{attribute 'linkalways'} 
{attribute 'no_explicit_call' := 'This FB is a CLASS and must be accessed using methods or properties'}
{attribute 'enable_dynamic_creation'}
FUNCTION_BLOCK Node_F_VN_AddToContainerElements_TcVnKeyPoint EXTENDS VisionNode
VAR
    stValue : _TcVnKeyPoint;
    ipContainer : _ITcVnContainer;
    hrPrev : _HRESULT(S_OK);
    hresult : _HRESULT(S_OK);
END_VAR

METHOD PUBLIC  Clone : I_Node
VAR
    pNode : POINTER TO Node_F_VN_AddToContainerElements_TcVnKeyPoint;
END_VAR
pNode := __NEW(Node_F_VN_AddToContainerElements_TcVnKeyPoint);
Clone := pNode^;
END_METHOD

METHOD FB_init : BOOL
VAR_INPUT
    bInitRetains : BOOL; // if TRUE, the retain variables are initialized (warm start / cold start)
    bInCopyCode : BOOL;  // if TRUE, the instance afterwards gets moved into the copy code (online change)
END_VAR
AddInput('stValue', stValue);
AddInput('ipContainer', ipContainer);
AddInput('hrPrev', hrPrev);
AddOutput('ipContainer', ipContainer);
AddOutput('hresult',hresult);
END_METHOD

METHOD PROTECTED OnExecute : HRESULT
hresult.Value := F_VN_AddToContainerElements_TcVnKeyPoint(
    stValue := stValue.Value,
    ipContainer := ipContainer.Value,
    hrPrev:= hrPrev.Value);
END_METHOD

METHOD PUBLIC PreExecutionCheck
VAR_INPUT
    Check : I_PreExecutionChecks;
END_VAR
Check.IsTrue(ipContainer.IsValid, 'ipContainer must be a valid container');
Check.IsTrue(ipContainer.HasType(TC_GLOBAL_CONST_LIST.ContainerType_Vector_TcVnKeyPoint), 'ipContainer contains incorrect type');
END_METHOD

END_FUNCTION_BLOCK

(* stored: Version 1.1.0.1, ProductVersion 3.1.4024.13
   POU Node_F_VN_AddToContainerElements_TcVnKeyPoint: Id {6e3b0a6c-2794-43ca-9f20-b43f5a6ce6cd}, SpecialFunc None
   Folder Constructor: Id {3ffa9107-90f1-47c6-8897-0875381fd3d9}
   Method Clone: Id {c6804d6d-485c-4786-ae2a-2958f9648dd4}
   Method FB_init: Id {7f42eba8-7316-4a11-8e1f-c000245f3363}
   Method OnExecute: Id {a69488e9-82ed-416d-abaa-ff13a16b610f}
   Method PreExecutionCheck: Id {9539a2f4-3b4a-4a16-8e6f-e4e5d30351e4} *)
